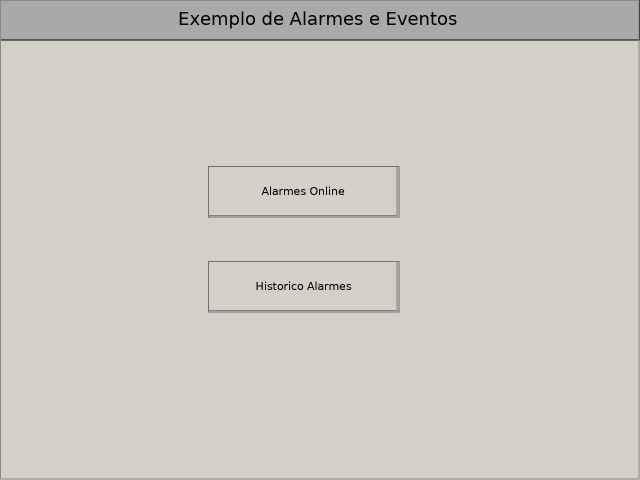
VISUALIZATION VISU_MAIN  // 640x480
    Button (208,261 191x51), "Historico Alarmes"
        OnMouseClick: change screen: VISU_EVENTS
    Rectangle (0,-1 640x41)
    Label (0,4 636x30), "Exemplo de Alarmes e Eventos"
    Button (208,166 191x51), "Alarmes Online"
        OnMouseClick: change screen: VISU_ALARMS
END_VISUALIZATION

(* stored: Version 1.1.0.1, ProductVersion 3.1.4024.12
   Visu VISU_MAIN: Id {57e258e5-f44b-4a4c-af4e-dd286d9b308f} *)
